(* CODESYS project Hackathon-Superviz.project

Project tree, tasks and I/O mapping:
  Device : CPX-CEC-C1-V3, Festo AG & Co. KG, order no. 3473128, version 3.5.7.37
      unmapped channels: Rotary switch
    application Application
      libraries: Standard, * (System)
      task MainTask (cyclic, interval t#20ms, priority 20) calls PLC_PRG
      program PLC_PRG [ST]
      global variables GVL
    PLC_Diagnosis : PLC-Diagnosis, Festo AG & Co. KG, version 3.5.4.1
    CPX_System : CPX_System, Festo AG & Co. KG, order no. 3473128, version 1.258
      CEC_C1_V3 : CEC-C1-V3, Festo AG & Co. KG, order no. 3473128, version 1.258
          settings:  = 0;  = 150810762677760;  = 839035072;  = 65535;  = 16885952;  = 13959208;  = 1f5d2989;  = 5
      _8DI_8DO : 8DI/8DO, Festo AG & Co. KG, order no. 526257, version 1.258
          settings:  = 0;  = 1;  = 1;  = 1;  = 1;  = 0;  = 1;  = 1;  = 0;  = 0;  = 0;  = 0;  = 0;  = 0;  = 0;  = 0;  = 0;  = 0;  = 0;  = 0;  = 0;  = 0;  = 0;  = 0;  = 0;  = 0;  = 0;  = 0;  = 0;  = 0;  = 0;  = 0;  = 0;  = 0;  = 0;  = 0;  = 0;  = 0;  = 0;  = 0;
             = 0;  = 0;  = 0;  = 0;  = 0;  = 0;  = 0;  = 0;  = 0;  = 0;  = 0;  = 0;  = 0;  = 0;  = 0;  = 0;  = 0;  = 0;  = 0;  = 0;  = 0;  = 0;  = 0;  = 0;  = 0;  = 0;  = 0;  = 0;  = 0;  = 0;  = 0;  = 0;  = 0;  = 0;  = 0;  = 0;  = 0;  = 0;  = 0;  = 0;
             = 576751027668385792;  = 'PI%i.0.0.1=1';  = 'PI%i.0.1.1=1';  = 'PI%i.0.2.1=1';  = 'PI%i.1.0.1=1';  = 'PI%i.1.1.1=0';  = 'PI%i.1.4.2=1';  = 'PI%i.1.6.2=1';  = 'PI%i.6.0.1=0';  = 'PI%i.6.1.1=0';  = 'PI%i.6.2.1=0';  = 'PI%i.6.3.1=0';  = 'PI%i.6.4.1=0';  = 'PI%i.6.5.1=0';  = 'PI%i.6.6.1=0';  = 'PI%i.6.7.1=0';  = dd4a6e5f;  = 6
          unmapped channels: Input 0, Output 0
      _8DI_8DO_1 : 8DI/8DO, Festo AG & Co. KG, order no. 526257, version 1.258
          settings:  = 0;  = 1;  = 1;  = 1;  = 1;  = 0;  = 1;  = 1;  = 0;  = 0;  = 0;  = 0;  = 0;  = 0;  = 0;  = 0;  = 0;  = 0;  = 0;  = 0;  = 0;  = 0;  = 0;  = 0;  = 0;  = 0;  = 0;  = 0;  = 0;  = 0;  = 0;  = 0;  = 0;  = 0;  = 0;  = 0;  = 0;  = 0;  = 0;  = 0;
             = 0;  = 0;  = 0;  = 0;  = 0;  = 0;  = 0;  = 0;  = 0;  = 0;  = 0;  = 0;  = 0;  = 0;  = 0;  = 0;  = 0;  = 0;  = 0;  = 0;  = 0;  = 0;  = 0;  = 0;  = 0;  = 0;  = 0;  = 0;  = 0;  = 0;  = 0;  = 0;  = 0;  = 0;  = 0;  = 0;  = 0;  = 0;  = 0;  = 0;
             = 576751027668385792;  = 'PI%i.0.0.1=1';  = 'PI%i.0.1.1=1';  = 'PI%i.0.2.1=1';  = 'PI%i.1.0.1=1';  = 'PI%i.1.1.1=0';  = 'PI%i.1.4.2=1';  = 'PI%i.1.6.2=1';  = 'PI%i.6.0.1=0';  = 'PI%i.6.1.1=0';  = 'PI%i.6.2.1=0';  = 'PI%i.6.3.1=0';  = 'PI%i.6.4.1=0';  = 'PI%i.6.5.1=0';  = 'PI%i.6.6.1=0';  = 'PI%i.6.7.1=0';  = dd4a6e61;  = 6
          unmapped channels: Input 0, Output 0
    Ethernet : Ethernet, 3S - Smart Software Solutions GmbH, version 3.5.10.0
      ModbusTCP_Slave_Device : ModbusTCP Slave Device, 3S - Smart Software Solutions GmbH, version 3.5.10.0
          settings: Unit-ID = 5
          unmapped channels: Inputs, Outputs
*)

// Device/Application/GVL
{attribute 'qualified_only'}
VAR_GLOBAL
	
//IHM
	//Entrada
	ihm_start	    AT	%IX2.0	:BOOL;  //Botão de start
	ihm_stop 		AT	%IX2.1	:BOOL;	//Botão de stop (NF)
	ihm_chave 		AT	%IX2.2	:BOOL;	//Chave auto/manual
	ihm_reset 		AT	%IX2.3	:BOOL;	//Botão de reset
	i4_ihm			AT	%IX2.4	:BOOL;	//Bit de saída 4 da IHM
	i5_ihm			AT	%IX2.5	:BOOL;	//Bit de saída 5 da IHM
	i6_ihm 			AT	%IX2.6	:BOOL;	//Bit de saída 6 da IHM
	i7_ihm			AT	%IX2.7	:BOOL;	//Bit de saída 7 da IHM	
	//Saída
	ihm_led_start   AT 	%QX1.0	:BOOL;
	ihm_led_reset   AT 	%QX1.1 	:BOOL;
	ihm_led_q1      AT 	%QX1.2 	:BOOL;
	ihm_led_q2      AT 	%QX1.3 	:BOOL;
	q4_ihm			AT	%QX1.4	:BOOL;	//Saída Q4 IHM
	q5_ihm			AT	%QX1.5	:BOOL;	//Saída Q5 IHM
	q6_ihm			AT	%QX1.6	:BOOL;	//Saída Q6 IHM
	q7_ihm   		AT	%QX1.7	:BOOL;	//Saída Q7 IHM

//SENSORES
	//Entrada
	s_inicial 		AT 	%IX1.0 	:BOOL; 	//Sensor de inicio
	s_atuador_b1 	AT 	%IX1.1	:BOOL;	//Sensor indutivo do atuador 1
	s_fim 			AT 	%IX1.2	:BOOL;  //Sensor de fim de rampa
	s_atuador_b2 	AT 	%IX1.3	:BOOL; 	//Sensor indutivo do atuador 2	
	s_barreira		AT 	%IX1.4	:BOOL;	//Sensor de barreira
	s_cor 			AT 	%IX1.5 	:BOOL;	//Sensor reflexivo
	s_indutivo 		AT 	%IX1.6 	:BOOL;	//Sensor indutivo presente na barreira
	
//ATUADORES 
	//Saída
	esteira_h 		AT	%QX0.0	:BOOL;	//Mover a esteira para frente
	atuador_b1	 	AT	%QX0.1	:BOOL;	//Aciona o pistão I
	atuador_b2	 	AT	%QX0.2	:BOOL;	//Aciona o pistão II
	atuador_p	 	AT	%QX0.3	:BOOL;	//Aciona o pistão I

//Bits - MODBUS 
	//Bits - Entrada (Holding registers)
	Stop  AT %IX4.0 : BOOL;
	Reset AT %IX4.1 : BOOL;
	Start AT %IX4.2 : BOOL;
	
	//Bits - Saida (Input registers)
	flag_preta  		AT %QX2.0 : BOOL;
	flag_prata  		AT %QX2.1 : BOOL;
	flag_vermelha  		AT %QX2.2 : BOOL;
	flag_robot 			AT %QX2.3 : BOOL;
END_VAR

// Device/Application/PLC_PRG
PROGRAM PLC_PRG
VAR
	steps : INT;
	
	timerq2_1: TON;
	IN_timerq2_1 : BOOL;
	timerq2_2 : TON;
	IN_timerq2_2 : BOOL;
	
	timer1 : TON;
	IN_timer1 : BOOL;
	timer_reset : TON; 
	IN_timer_reset : BOOL; 
	timerEndProcess : TON;
	IN_timerEndProcess : BOOL;
	
	
	flag_reset: BOOL;
	flag_start: BOOL;
	flag_prod : BOOL;
	flag_endprocess : BOOL;
	flag_robot : BOOL;
	flag_preta : BOOL;
	flag_prata : BOOL;
	flag_vermelha : BOOL;
	
	//Flag controle de processo
	station_stop_state : BOOL;
	station_reset_state : BOOL;		
	station_start_state : BOOL;
END_VAR

//Programa estação 5 Central Ciberconectividade - 30/09/2024
//Luizinho - =) 

//Bit association
gvl.flag_preta := flag_preta; 
gvl.flag_prata := flag_prata; 
gvl.flag_vermelha := flag_vermelha; 
gvl.flag_robot := flag_robot; 


//Configuração dos timer
	//Timers de controle
	timer1(IN:= IN_timer1, PT:=T#2S);
	timerEndProcess(IN:= IN_timerEndProcess, PT:=T#5S);

	timer_reset (IN:= IN_timer_reset, PT:=T#0.8S);
	
	//Timer de Blynk Leds	
	timerq2_1(IN:= IN_timerq2_1, PT:=T#0.3S);
	timerq2_2 (IN:= IN_timerq2_2, PT:=T#0.3S);

//--------------------Pisca-pisca Q2
IF timerq2_1.Q THEN
	gvl.ihm_led_q2 := TRUE;
	IN_timerq2_1 := FALSE;
	IN_timerq2_2 := TRUE;
END_IF
IF timerq2_2.Q THEN
	gvl.ihm_led_q2 := FALSE; 
	IN_timerq2_2 := FALSE;
	IN_timerq2_1 := TRUE;
END_IF

//--------------------Stop Botton
IF NOT gvl.ihm_stop OR gvl.Stop THEN
	station_stop_state := TRUE;
	station_reset_state := FALSE;
	station_start_state := FALSE;
	gvl.atuador_b1 := FALSE;
	gvl.atuador_b2 := FALSE;
	gvl.atuador_p := FALSE;
	gvl.esteira_h  := FALSE;
	gvl.ihm_led_q2 := FALSE;
	gvl.ihm_led_q1 := FALSE;
	gvl.ihm_led_reset := TRUE;
	gvl.ihm_led_start := FALSE;
	IN_timer1 := FALSE;
	IN_timerEndProcess := FALSE;
	IN_timer_reset := FALSE;
	IN_timerq2_1 := FALSE;
	IN_timerq2_2 := FALSE;
	flag_reset := TRUE;
	flag_start := FALSE;
	flag_prod := FALSE;	
	flag_preta := FALSE;
	flag_prata := FALSE;
	flag_vermelha := FALSE;
	flag_endprocess := FALSE;
	steps := 400;
END_IF

//--------------------Reset Botton
IF (gvl.ihm_reset OR gvl.Reset) AND NOT flag_start AND flag_reset THEN
	station_stop_state := FALSE;
	station_reset_state := TRUE;
	station_start_state := FALSE;
	gvl.ihm_led_q1 := TRUE;
	gvl.ihm_led_reset := FALSE;
	gvl.ihm_led_start := TRUE;
	gvl.atuador_b1 := TRUE;
	gvl.atuador_b2 := TRUE;
	IN_timer_reset := TRUE;
	flag_reset := FALSE;
	flag_start := TRUE;
	steps := 0;
END_IF

IF timer_reset.Q THEN
	IN_timer_reset := FALSE;
	gvl.atuador_b1 := FALSE;
	gvl.atuador_b2 := FALSE;
END_IF

//--------------------Start Botton
IF (gvl.Start OR gvl.ihm_start) AND flag_start THEN
	station_stop_state := FALSE;
	station_reset_state := FALSE;
	station_start_state := TRUE;
	gvl.ihm_led_start := FALSE;
	flag_start := FALSE;
	flag_prod := TRUE;
END_IF

IF steps = 0 AND flag_prod AND NOT flag_start THEN
	gvl.q4_ihm := TRUE;
	steps := 1;
END_IF

IF steps = 1 AND gvl.s_inicial THEN
	gvl.esteira_h := TRUE;
	gvl.q4_ihm := FALSE;
	IN_timerq2_1 := TRUE;
	steps := 2;
END_IF

IF steps = 2 THEN 
	IN_timer1 := TRUE;
	steps := 3;
END_IF

IF steps = 3 AND timer1.Q AND gvl.s_cor AND gvl.s_indutivo THEN // Peça Prata
	gvl.atuador_p := TRUE;
	gvl.atuador_b1 := TRUE;
	flag_prata := TRUE;

	steps := 4;
END_IF

IF steps = 3 AND timer1.Q AND gvl.s_cor AND NOT gvl.s_indutivo THEN // Peça rosa
	gvl.atuador_p := TRUE;
	gvl.atuador_b2 := TRUE;
	flag_vermelha := TRUE;
	steps := 4;
END_IF

IF steps = 3 AND timer1.Q AND NOT gvl.s_cor AND NOT gvl.s_indutivo THEN // Peça preta
	gvl.atuador_p := TRUE;
	flag_preta := TRUE;
	steps := 4;
END_IF

IF steps = 4 AND gvl.s_fim THEN
	gvl.esteira_h := FALSE;
	gvl.atuador_b1 := FALSE;
	gvl.atuador_b2 := FALSE;
	gvl.atuador_p := FALSE;
	gvl.ihm_led_q2 := FALSE;
	IN_timer1 := FALSE;
	IN_timerq2_1 := FALSE;
	IN_timerq2_2 := FALSE;
	flag_endprocess := TRUE;
	IN_timerEndProcess := TRUE;
	steps := 0;
END_IF

IF gvl.i4_ihm THEN
	flag_robot := TRUE;
ELSE
	flag_robot := FALSE;
END_IF
IF flag_endprocess AND timerEndProcess.Q THEN
	IN_timerEndProcess := FALSE;
	flag_preta := FALSE;
	flag_prata := FALSE;
	flag_vermelha := FALSE;
END_IF

END_PROGRAM
